VAR_GLOBAL
END_VAR

(* stored: Version 1.1.0.1, ProductVersion 3.1.0.19
   GVL MER_CmdState: Id {45905dd6-ef8e-419f-be60-bfa14a24c19d} *)
